Staubli VAL3: SimpleMessage.dtx

public CommType commType
  [0]
    num nRequest = 2
    num nResponse = 3
public ReplyType replyType
  [0]
    num nSuccess = 1
    num nFailure = 2
